// TIA Portal V20 export
DATA_BLOCK "LBP_PIServices"   // DB16
TITLE = PI Services / Services PI
// Interface for LBP_ReqPIService [FB7], contains definitions for all available PI services. / L'interface pour LBP_ReqPIService [FB7] contient des définitions pour tous les services PI disponibles.
   VAR
      SELECT : Struct
         PIName : String[10] := '_N_SELECT';
         p01 : Byte := BYTE#16#03;   // Area / Unit / Zone/unité
         p02 : Char := '2';   // Area identifier / Identificateur de zone
         p11 : Byte := BYTE#16#FD;   // Path name / Nom de chemin
         p12 : Byte := BYTE#16#13;   // Add string with arbitrary number of odd numbers / Ajouter une chaîne contenant un nombre quelconque de nombres impairs
         p21 : Byte := BYTE#16#FE;   // Program name / Nom de programme
         p22 : Byte := BYTE#16#13;   // Add string with arbitrary number of odd numbers / Ajouter une chaîne contenant un nombre quelconque de nombres impairs
      END_STRUCT;
      ASUP : Struct
         PIName : String[10] := '_N_ASUP__';
         p01 : Byte := BYTE#16#03;   // Area / Unit / Zone/unité
         p02 : Char := '2';   // Area identifier / Identificateur de zone
         p11 : Byte := BYTE#16#03;   // Interrupt number / Numéro d'interruption
         p12 : Byte := BYTE#16#05;   // Int from WORD specification / INT de spécification WORD
         p21 : Byte := BYTE#16#03;   // Priority / Priorité
         p22 : Byte := BYTE#16#05;   // Int from WORD specification / INT de spécification WORD
         p31 : Byte := BYTE#16#01;   // Liftfast
         p32 : Byte := BYTE#16#05;   // Int from WORD specification / INT de spécification WORD
         p41 : Byte := BYTE#16#01;   // Blocksync
         p42 : Byte := BYTE#16#05;   // Int from WORD specification / INT de spécification WORD
         p51 : Byte := BYTE#16#FD;   // Path name / Nom de chemin
         p52 : Byte := BYTE#16#13;   // Add string with arbitrary number of odd numbers / Ajouter une chaîne contenant un nombre quelconque de nombres impairs
         p61 : Byte := BYTE#16#FE;   // Program name / Nom de programme
         p62 : Byte := BYTE#16#13;   // Add string with arbitrary number of odd numbers / Ajouter une chaîne contenant un nombre quelconque de nombres impairs
      END_STRUCT;
      FINDBL : Struct
         PIName : String[10] := '_N_FINDBL';
         p01 : Byte := BYTE#16#03;   // Area / Unit / Zone/unité
         p02 : Char := '2';
         p11 : Byte := BYTE#16#01;   // Preprocessing mode / Mode de prétraitement
         p12 : Byte := BYTE#16#04;   // Word from WORD specification / Mot depuis spécification WORD
      END_STRUCT;
      SETUFR : Struct
         PIName : String[10] := '_N_SETUFR';
         p01 : Byte := BYTE#16#03;   // Area / Unit / Zone/unité
         p02 : Char := '2';
      END_STRUCT;
      CANCEL : Struct
         PIName : String[10] := '_N_CANCEL';
         p01 : Byte := BYTE#16#03;   // Area / Unit / Zone/unité
         p02 : Char := '0';
      END_STRUCT;
      DELETO : Struct
         PIName : String[10] := '_N_DELETO';
         p01 : Byte := BYTE#16#03;   // Area / Unit / Zone/unité
         p02 : Char := '4';
         p11 : Byte := BYTE#16#05;   // T number / Numéro d'outil
         p12 : Byte := BYTE#16#05;   // Int from WORD specification / INT de spécification WORD
      END_STRUCT;
      CREATO : Struct
         PIName : String[10] := '_N_CREATO';
         p01 : Byte := BYTE#16#03;   // Area / Unit / Zone/unité
         p02 : Char := '4';
         p11 : Byte := BYTE#16#05;   // T number / Numéro d'outil
         p12 : Byte := BYTE#16#05;   // Int from WORD specification / INT de spécification WORD
      END_STRUCT;
      CREACE : Struct
         PIName : String[10] := '_N_CREACE';
         p01 : Byte := BYTE#16#03;   // Area / Unit / Zone/unité
         p02 : Char := '4';
         p11 : Byte := BYTE#16#05;   // T number / Numéro d'outil
         p12 : Byte := BYTE#16#05;   // Int from WORD specification / INT de spécification WORD
      END_STRUCT;
      TMCRTO : Struct
         PIName : String[10] := '_N_TMCRTO';
         p01 : Byte := BYTE#16#03;   // Area / Unit / Zone/unité
         p02 : Char := '4';
         p11 : Byte := BYTE#16#20;   // Tool identifier, add blank / Identifiant d'outil, ajouter espace
         p12 : Byte := BYTE#16#13;   // String identifier! / Identifiant de chaîne.
         p21 : Byte := BYTE#16#05;   // T number / Numéro d'outil
         p22 : Byte := BYTE#16#05;   // Int from WORD specification / INT de spécification WORD
         p31 : Byte := BYTE#16#05;   // Duplo number / Numéro d'outil frère
         p32 : Byte := BYTE#16#05;   // Int from WORD specification / INT de spécification WORD
      END_STRUCT;
      TMFDPL : Struct
         PIName : String[10] := '_N_TMFDPL';
         p01 : Byte := BYTE#16#03;   // Area / Unit / Zone/unité
         p02 : Char := '4';
         p11 : Byte := BYTE#16#05;   // T number / Numéro d'outil
         p12 : Byte := BYTE#16#05;   // Int from WORD specification / INT de spécification WORD
         p21 : Byte := BYTE#16#05;   // Location number (target) / Numéro d'emplacement (cible)
         p22 : Byte := BYTE#16#05;   // Int from WORD specification / INT de spécification WORD
         p31 : Byte := BYTE#16#05;   // Magazine number (target) / Numéro de magasin (cible)
         p32 : Byte := BYTE#16#05;   // Int from WORD specification / INT de spécification WORD
         p41 : Byte := BYTE#16#05;   // Location number (reference) / Numéro d'emplacement (référence)
         p42 : Byte := BYTE#16#05;   // Int from WORD specification / INT de spécification WORD
         p51 : Byte := BYTE#16#05;   // Magazine number (reference) / ID Numéro de magasin (référence)
         p52 : Byte := BYTE#16#05;   // Int from WORD specification / INT de spécification WORD
      END_STRUCT;
      TMMVTL : Struct
         PIName : String[10] := '_N_TMMVTL';
         p01 : Byte := BYTE#16#03;   // Area / Unit / Zone/unité
         p02 : Char := '4';
         p11 : Byte := BYTE#16#05;   // T number / Numéro d'outil
         p12 : Byte := BYTE#16#05;   // Int from WORD specification / INT de spécification WORD
         p21 : Byte := BYTE#16#05;   // Location number (source) / Numéro d'emplacement (source)
         p22 : Byte := BYTE#16#05;   // Int from WORD specification / INT de spécification WORD
         p31 : Byte := BYTE#16#05;   // Magazine number (source) / Numéro de magasin (source)
         p32 : Byte := BYTE#16#05;   // Int from WORD specification / INT de spécification WORD
         p41 : Byte := BYTE#16#05;   // Location number (target) / Numéro d'emplacement (cible)
         p42 : Byte := BYTE#16#05;   // Int from WORD specification / INT de spécification WORD
         p51 : Byte := BYTE#16#05;   // Magazine number (target) / Numéro de magasin (cible)
         p52 : Byte := BYTE#16#05;   // Int from WORD specification / INT de spécification WORD
      END_STRUCT;
      TMPCIT : Struct
         PIName : String[10] := '_N_TMPCIT';
         p01 : Byte := BYTE#16#03;   // Area / Unit / Zone/unité
         p02 : Char := '4';
         p11 : Byte := BYTE#16#03;   // Spindle number / Numéro de broche
         p12 : Byte := BYTE#16#05;   // Int from WORD specification / INT de spécification WORD
         p21 : Byte := BYTE#16#05;   // Increment value / Incrément valeur
         p22 : Byte := BYTE#16#05;   // Int from WORD specification / INT de spécification WORD
      END_STRUCT;
      TMPOSM : Struct
         PIName : String[10] := '_N_TMPOSM';
         p01 : Byte := BYTE#16#03;   // Area / Unit / Zone/unité
         p02 : Char := '4';
         p11 : Byte := BYTE#16#05;   // T number / Numéro d'outil
         p12 : Byte := BYTE#16#05;   // Int from WORD specification / INT de spécification WORD
         p21 : Byte := BYTE#16#20;   // Tool identifier, add blank / Identificateur d'outil, ajouter espace
         p22 : Byte := BYTE#16#13;   // String identifier! / Identifiant de chaîne.
         p31 : Byte := BYTE#16#05;   // Duplo number / Numéro d'outil frère
         p32 : Byte := BYTE#16#05;   // Int from WORD specification / INT de spécification WORD
         p41 : Byte := BYTE#16#05;   // Location number (source) / Numéro d'emplacement (source)
         p42 : Byte := BYTE#16#05;   // Int from WORD specification / INT de spécification WORD
         p51 : Byte := BYTE#16#05;   // Magazine number (source) / Numéro de magasin (source)
         p52 : Byte := BYTE#16#05;   // Int from WORD specification / INT de spécification WORD
         p61 : Byte := BYTE#16#05;   // Location number (target) / Numéro d'emplacement (cible)
         p62 : Byte := BYTE#16#05;   // Int from WORD specification / INT de spécification WORD
         p71 : Byte := BYTE#16#05;   // Magazine number (target) / Numéro de magasin (cible)
         p72 : Byte := BYTE#16#05;   // Int from WORD specification / INT de spécification WORD
      END_STRUCT;
      DIGION : Struct
         PIName : String[10] := '_N_DIGION';
         p01 : Byte := BYTE#16#03;   // Area / Unit / Zone/unité
         p02 : Char := '2';
      END_STRUCT;
      DIGIOF : Struct
         PIName : String[10] := '_N_DIGIOF';
         p01 : Byte := BYTE#16#03;   // Area / Unit / Zone/unité
         p02 : Char := '2';
      END_STRUCT;
      CONFIG : Struct
         PIName : String[10] := '_N_CONFIG';
         p01 : Byte := BYTE#16#03;   // Area / Unit / Zone/unité
         p02 : Char := '0';
         p11 : Byte := BYTE#16#02;   // Classification
         p12 : Byte := BYTE#16#04;   // Int from WORD specification / INT de spécification WORD
      END_STRUCT;
      LOGIN : Struct
         PIName : String[10] := '_N_LOGIN_';
         p01 : Byte := BYTE#16#03;   // Area / Unit / Zone/unité
         p02 : Char := '0';
         p11 : Byte := BYTE#16#20;   // Password (8 to 32 characters) / Mot de passe (8 à 32 caractères)
         p12 : Byte := BYTE#16#13;   // String identifier! / Identifiant de chaîne.
      END_STRUCT;
      LOGOUT : Struct
         PIName : String[10] := '_N_LOGOUT';
         p01 : Byte := BYTE#16#03;   // Area / Unit / Zone/unité
         p02 : Char := '0';
      END_STRUCT;
      MMCSEM : Struct
         PIName : String[10] := '_N_MMCSEM';
         p01 : Byte := BYTE#16#03;   // Area / Unit / Zone/unité
         p02 : Char := '2';
         p11 : Byte := BYTE#16#03;   // Function number / Numéro de fonction
         p12 : Byte := BYTE#16#05;   // Int from WORD specification / INT de spécification WORD
         p21 : Byte := BYTE#16#01;   // Semaphore value / Valeur sémaphore
         p22 : Byte := BYTE#16#05;   // Int from WORD specification / INT de spécification WORD
      END_STRUCT;
      DELECE : Struct
         PIName : String[10] := '_N_DELECE';
         p01 : Byte := BYTE#16#03;   // Area / Unit / Zone/unité
         p02 : Char := '4';
         p11 : Byte := BYTE#16#05;   // T number / Numéro d'outil
         p12 : Byte := BYTE#16#05;   // Int from WORD specification / INT de spécification WORD
         p21 : Byte := BYTE#16#05;   // D number / Numéro D
         p22 : Byte := BYTE#16#05;   // Int from WORD specification / INT de spécification WORD
      END_STRUCT;
      CRCEDN : Struct
         PIName : String[10] := '_N_CRCEDN';
         p01 : Byte := BYTE#16#03;   // Area / Unit / Zone/unité
         p02 : Char := '4';
         p11 : Byte := BYTE#16#05;   // T number / Numéro d'outil
         p12 : Byte := BYTE#16#05;   // Int from WORD specification / INT de spécification WORD
         p21 : Byte := BYTE#16#05;   // D number / Numéro D
         p22 : Byte := BYTE#16#05;   // Int from WORD specification / INT de spécification WORD
      END_STRUCT;
      TSEARC : Struct
         PIName : String[10] := '_N_TSEARC';
         p01 : Byte := BYTE#16#03;   // Area / Unit / Zone/unité
         p02 : Char := '4';
         p11 : Byte := BYTE#16#05;   // from: Magazine number / de : numéro de magasin
         p12 : Byte := BYTE#16#05;   // Int from WORD specification / INT de spécification WORD
         p21 : Byte := BYTE#16#05;   // from: Location number / de : numéro d'emplacement
         p22 : Byte := BYTE#16#05;   // Int from WORD specification / INT de spécification WORD
         p31 : Byte := BYTE#16#05;   // up to: Magazine number / à : numéro de magasin
         p32 : Byte := BYTE#16#05;   // Int from WORD specification / INT de spécification WORD
         p41 : Byte := BYTE#16#05;   // up to: Location number / à : numéro d'emplacement
         p42 : Byte := BYTE#16#05;   // Int from WORD specification / INT de spécification WORD
         p51 : Byte := BYTE#16#05;   // Number of reference magazine / Numéro du magasin de référence
         p52 : Byte := BYTE#16#05;   // Int from WORD specification / INT de spécification WORD
         p61 : Byte := BYTE#16#05;   // Number of reference location / Numéro de l'emplacement de référence
         p62 : Byte := BYTE#16#05;   // Int from WORD specification / INT de spécification WORD
         p71 : Byte := BYTE#16#01;   // Search direction / Sens de recherche
         p72 : Byte := BYTE#16#05;   // Int from WORD specification / INT de spécification WORD
         p81 : Byte := BYTE#16#01;   // Tool properties / Caractéristiques de l'outil
         p82 : Byte := BYTE#16#05;   // Int from WORD specification / INT de spécification WORD
      END_STRUCT;
      TMFPBP : Struct
         PIName : String[10] := '_N_TMFPBP';
         p01 : Byte := BYTE#16#03;   // Area / Unit / Zone/unité
         p02 : Char := '4';
         p11 : Byte := BYTE#16#05;   // from: Magazine number / de : numéro de magasin
         p12 : Byte := BYTE#16#05;   // Int from WORD specification / INT de spécification WORD
         p21 : Byte := BYTE#16#05;   // from: Location number / de : numéro d'emplacement
         p22 : Byte := BYTE#16#05;   // Int from WORD specification / INT de spécification WORD
         p31 : Byte := BYTE#16#05;   // up to: Magazine number / à : numéro de magasin
         p32 : Byte := BYTE#16#05;   // Int from WORD specification / INT de spécification WORD
         p41 : Byte := BYTE#16#05;   // up to: Location number / à : numéro d'emplacement
         p42 : Byte := BYTE#16#05;   // Int from WORD specification / INT de spécification WORD
         p51 : Byte := BYTE#16#05;   // Number of reference magazine / Numéro du magasin de référence
         p52 : Byte := BYTE#16#05;   // Int from WORD specification / INT de spécification WORD
         p61 : Byte := BYTE#16#05;   // Number of reference location / Numéro de l'emplacement de référence
         p62 : Byte := BYTE#16#05;   // Int from WORD specification / INT de spécification WORD
         p71 : Byte := BYTE#16#05;   // Number of locations to the left / Nombre d'emplacements vers la gauche
         p72 : Byte := BYTE#16#05;   // Int from WORD specification / INT de spécification WORD
         p81 : Byte := BYTE#16#05;   // Number of locations to the right / Nombre d'emplacements vers la droite
         p82 : Byte := BYTE#16#05;   // Int from WORD specification / INT de spécification WORD
         p91 { ExternalVisible := 'False'} : Byte := BYTE#16#05;   // Number of locations above / Nombre d'emplacements vers le haut
         p92 : Byte := BYTE#16#05;   // Int from WORD specification / INT de spécification WORD
         pa1 : Byte := BYTE#16#05;   // Number of locations below / Nombre d'emplacements vers le bas
         pa2 : Byte := BYTE#16#05;   // Int from WORD specification / INT de spécification WORD
         pb1 : Byte := BYTE#16#05;   // Location type index / Type d'emplacement Indice
         pb2 : Byte := BYTE#16#05;   // Int from WORD specification / INT de spécification WORD
         pc1 : Byte := BYTE#16#05;   // Search direction / Sens de recherche
         pc2 : Byte := BYTE#16#05;   // Int from WORD specification / INT de spécification WORD
      END_STRUCT;
      NCRES : Struct
         PIName : String[10] := '_N_IBN_SS';
         p01 : Byte := BYTE#16#03;   // Area / Unit / Zone/unité
         p02 : Char := 'K';
         p11 : Byte := BYTE#16#01;   // Classification
         p12 : Byte := BYTE#16#04;   // WORD specification / Spécification WORD
      END_STRUCT;
      TMRASS : Struct
         PIName : String[10] := '_N_TMRASS';
         p01 : Byte := BYTE#16#03;   // Area / Unit / Zone/unité
         p02 : Char := '4';
      END_STRUCT;
      TRESMO : Struct
         PIName : String[10] := '_N_TRESMO';
         p01 : Byte := BYTE#16#03;   // Area / Unit / Zone/unité
         p02 : Char := '4';
         p11 : Byte := BYTE#16#05;   // Tool number / Numéro d'outil
         p12 : Byte := BYTE#16#05;   // Int from WORD specification / INT de spécification WORD
         p21 : Byte := BYTE#16#05;   // D number / Numéro D
         p22 : Byte := BYTE#16#05;   // Int from WORD specification / INT de spécification WORD
         p31 : Byte := BYTE#16#05;   // Monitoring type / Type de surveillance
         p32 : Byte := BYTE#16#05;   // Int from WORD specification / INT de spécification WORD
      END_STRUCT;
      TMGETT : Struct
         PIName : String[10] := '_N_TMGETT';
         p01 : Byte := BYTE#16#03;   // Area / Unit / Zone/unité
         p02 : Char := '4';
         p11 : Byte := BYTE#16#20;   // Tool identifier, add blank / Identifiant d'outil, ajouter espace
         p12 : Byte := BYTE#16#13;   // String identifier! / Identifiant de chaîne.
         p21 : Byte := BYTE#16#05;   // Duplo number / Numéro d'outil frère
         p22 : Byte := BYTE#16#05;   // Int from WORD specification / INT de spécification WORD
      END_STRUCT;
      SETUDT : Struct
         PIName : String[10] := '_N_SETUDT';
         p01 : Byte := BYTE#16#03;   // Area / Unit / Zone/unité
         p02 : Char := '2';
         p11 : Byte := BYTE#16#03;   // UserDataType
         p12 : Byte := BYTE#16#04;   // WORD specification / Spécification WORD
         p21 : Byte := BYTE#16#05;   // ind1
         p22 : Byte := BYTE#16#04;   // WORD specification / Spécification WORD
         p31 : Byte := BYTE#16#05;   // ind2
         p32 : Byte := BYTE#16#04;   // WORD specification / Spécification WORD
      END_STRUCT;
      TMCRMT : Struct
         PIName : String[10] := '_N_TMCRMT';
         p01 : Byte := BYTE#16#03;   // Area / Unit / Zone/unité
         p02 : Char := '4';
         p11 : Byte := BYTE#16#20;   // Multitool identifier, insert blanks / Identifiant Multitool, ajouter espace
         p12 : Byte := BYTE#16#13;   // String identifier! / Identifiant de chaîne.
         p21 : Byte := BYTE#16#05;   // Reserved / Réservé
         p22 : Byte := BYTE#16#05;   // Int from WORD specification / INT de spécification WORD
         p31 : Byte := BYTE#16#05;   // Multitool number / Numéro Multitool
         p32 : Byte := BYTE#16#05;   // Int from WORD specification / INT de spécification WORD
         p41 : Byte := BYTE#16#03;   // Number of Multitool locations / Nombre d'emplacements Multitool
         p42 : Byte := BYTE#16#05;   // Int from WORD specification / INT de spécification WORD
         p51 : Byte := BYTE#16#01;   // Type of distance coding / Type de codage de distance
         p52 : Byte := BYTE#16#05;   // Int from WORD specification / INT de spécification WORD
      END_STRUCT;
      TMDLMT : Struct
         PIName : String[10] := '_N_TMDLMT';
         p01 : Byte := BYTE#16#03;   // Area / Unit / Zone/unité
         p02 : Char := '4';
         p11 : Byte := BYTE#16#20;   // Multitool identifier, insert blanks / Identifiant Multitool, ajouter espace
         p12 : Byte := BYTE#16#13;   // String identifier! / Identifiant de chaîne.
         p21 : Byte := BYTE#16#05;   // Reserved / Réservé
         p22 : Byte := BYTE#16#05;   // Int from WORD specification / INT de spécification WORD
         p31 : Byte := BYTE#16#05;   // Multitool number / Numéro Multitool
         p32 : Byte := BYTE#16#05;   // Int from WORD specification / INT de spécification WORD
         p41 : Byte := BYTE#16#01;   // Delete included tools / Supprimer les outils contenus
         p42 : Byte := BYTE#16#05;   // Int from WORD specification / INT de spécification WORD
      END_STRUCT;
      POSMT : Struct
         PIName : String[10] := '_N_POSMT_';
         p01 : Byte := BYTE#16#03;   // Area / Unit / Zone/unité
         p02 : Char := '4';
         p11 : Byte := BYTE#16#03;   // Number of toolholder / Numéro du porte-outil
         p12 : Byte := BYTE#16#05;   // Int from WORD specification / INT de spécification WORD
         p21 : Byte := BYTE#16#05;   // Tool number / Numéro d'outil
         p22 : Byte := BYTE#16#05;   // Int from WORD specification / INT de spécification WORD
         p31 : Byte := BYTE#16#20;   // Tool number, add blank / Identificateur d'outil, ajouter espace
         p32 : Byte := BYTE#16#13;   // String identifier! / Identifiant de chaîne.
         p41 : Byte := BYTE#16#05;   // Duplo number / Numéro d'outil frère
         p42 : Byte := BYTE#16#05;   // Int from WORD specification / INT de spécification WORD
         p51 : Byte := BYTE#16#03;   // Multitool place number / Numéro d'emplacement Multitool
         p52 : Byte := BYTE#16#05;   // Int from WORD specification / INT de spécification WORD
      END_STRUCT;
      FDPLMT : Struct
         PIName : String[10] := '_N_FDPLMT';
         p01 : Byte := BYTE#16#03;   // Area / Unit / Zone/unité
         p02 : Char := '4';
         p11 : Byte := BYTE#16#05;   // Tool number / Numéro d'outil
         p12 : Byte := BYTE#16#05;   // Int from WORD specification / INT de spécification WORD
         p21 : Byte := BYTE#16#20;   // Tool number, add blank / Identificateur d'outil, ajouter espace
         p22 : Byte := BYTE#16#13;   // String identifier! / Identifiant de chaîne.
         p31 : Byte := BYTE#16#05;   // Duplo number / Numéro d'outil frère
         p32 : Byte := BYTE#16#05;   // Int from WORD specification / INT de spécification WORD
         p41 : Byte := BYTE#16#05;   // Multitool number / Numéro Multitool
         p42 : Byte := BYTE#16#05;   // Int from WORD specification / INT de spécification WORD
         p51 : Byte := BYTE#16#03;   // Multitool place number / Numéro d'emplacement Multitool
         p52 : Byte := BYTE#16#05;   // Int from WORD specification / INT de spécification WORD
      END_STRUCT;
      RETRAC : Struct
         PIName : String[10] := '_N_RETRAC';
         p01 : Byte := BYTE#16#03;   // Area / Unit / Zone/unité
         p02 : Char := '2';
         p11 : Byte := BYTE#16#03;   // Geometry axis / Axe géométrique
         p12 : Byte := BYTE#16#04;   // WORD specification / Spécification WORD
         p21 : Byte := BYTE#16#05;   // Parameter2 / Paramètre2
         p22 : Byte := BYTE#16#04;   // WORD specification / Spécification WORD
      END_STRUCT;
   END_VAR
BEGIN
END_DATA_BLOCK
